FUNCTION_BLOCK FB_Tool EXTENDS FB_Base
VAR_INPUT
	sOpen: Skill_Greifer_open;
END_VAR
VAR_OUTPUT
	visStatus: stVisStatusTool;
END_VAR
VAR
END_VAR

ACTION CYCLIC_TOOL:
CYCLIC_BASE();


//VISSTATUS
//TODO

// GO INTO GREIFER.... INSTANCE OF THIS FB //todo
pA_Skills[1]:=ADR(sOpen);
sOpen(pTool:=THIS,pin:=9);
END_ACTION

METHOD PROTECTED onActivate : eResult
onActivate := eResult.SUCCESS;
      RETURN;
      // ---- Init ----
_transitionresult:=eResult.None;



// ---- Change ----

// _mode:= eMode.Automatic;




// ---- Check ----
_transitionresult := eResult.SUCCESS;


// ---- Change State ----
IF _transitionresult= eResult.SUCCESS THEN
	State:=eState.Active;
ELSIF _transitionresult= eResult.FAILURE THEN
	State:=eState.Inactive;
ELSIF _transitionresult= eResult.ERROR THEN
	State:=eState.ErrorProcessing;
ELSE
	ADSLOGSTR(ADSLOG_MSGTYPE_WARN,'Transitionresult from onActivate is None','');
END_IF
END_METHOD

METHOD PROTECTED onCleanup : eResult
onCleanup := eResult.SUCCESS;
      RETURN;
      // ---- Init ----
_transitionresult:=eResult.None;



// ---- Change ----

// _mode:= eMode.Manual;




// ---- Check ----
_transitionresult := eResult.SUCCESS;


// ---- Change State ----
IF _transitionresult= eResult.SUCCESS THEN
	State:=eState.Unconfigured;
ELSIF _transitionresult= eResult.FAILURE THEN
	ADSLOGSTR(ADSLOG_MSGTYPE_WARN,'Transitionresult from onCleanup is FAILURE ','');
ELSIF _transitionresult= eResult.ERROR THEN
	State:=eState.ErrorProcessing;
ELSE
	ADSLOGSTR(ADSLOG_MSGTYPE_WARN,'Transitionresult from onCleanup is NONE','');
END_IF
END_METHOD

METHOD PROTECTED onConfigure : eResult
onConfigure := eResult.SUCCESS;
      RETURN;
      // ---- Init ----
_transitionresult:=eResult.None;



// ---- Change ----

// _mode:= eMode.Manual;




// ---- Check ----
_transitionresult := eResult.SUCCESS;


// ---- Change State ----
IF _transitionresult= eResult.SUCCESS THEN
	State:=eState.Inactive;
ELSIF _transitionresult= eResult.FAILURE THEN
	State:=eState.Unconfigured;
ELSIF _transitionresult= eResult.ERROR THEN
	State:=eState.ErrorProcessing;
ELSE
	ADSLOGSTR(ADSLOG_MSGTYPE_WARN,'Transitionresult from onConfigure is None','');
END_IF
END_METHOD

METHOD PROTECTED onDeactivate : eResult
onDeactivate := eResult.SUCCESS;
      RETURN;
      // ---- Init ----
_transitionresult:=eResult.None;



// ---- Change ----

// _mode:= eMode.Manual;




// ---- Check ----
_transitionresult := eResult.SUCCESS;


// ---- Change State ----
IF _transitionresult= eResult.SUCCESS THEN
	State:=eState.Inactive;
ELSIF _transitionresult= eResult.FAILURE THEN
	ADSLOGSTR(ADSLOG_MSGTYPE_WARN,'Transitionresult from onDeactivate is FAILURE','');
ELSIF _transitionresult= eResult.ERROR THEN
	State:=eState.ErrorProcessing;
ELSE
	ADSLOGSTR(ADSLOG_MSGTYPE_WARN,'Transitionresult from onDeactivate is None','');
END_IF
END_METHOD

METHOD PROTECTED onError : eResult
onError := eResult.SUCCESS;
      RETURN;
      // ---- Init ----
_transitionresult:=eResult.None;



// ---- Change ----

// _mode:= eMode.Manual;




// ---- Check ----
_transitionresult := eResult.SUCCESS;


// ---- Change State ----
IF _transitionresult= eResult.SUCCESS THEN
	State:=eState.Unconfigured;
ELSIF _transitionresult= eResult.FAILURE THEN
	State:=eState.Finalized;
ELSIF _transitionresult= eResult.ERROR THEN
	ADSLOGSTR(ADSLOG_MSGTYPE_WARN,'Transitionresult from onError is Error','');
ELSE
	ADSLOGSTR(ADSLOG_MSGTYPE_WARN,'Transitionresult from onError is None','');
END_IF
END_METHOD

METHOD PROTECTED onShutdown : eResult
onShutdown := eResult.SUCCESS;
      RETURN;
      // ---- Init ----
_transitionresult:=eResult.None;



// ---- Change ----

// _mode:= eMode.Manual;




// ---- Check ----
_transitionresult := eResult.SUCCESS;


// ---- Change State ----
IF _transitionresult= eResult.SUCCESS THEN
	State:=eState.Finalized;
ELSIF _transitionresult= eResult.FAILURE THEN
	ADSLOGSTR(ADSLOG_MSGTYPE_WARN,'Transitionresult from onShutdown is FAILURE','');
ELSIF _transitionresult= eResult.ERROR THEN
	State:=eState.ErrorProcessing;
ELSE
	ADSLOGSTR(ADSLOG_MSGTYPE_WARN,'Transitionresult from onShutdown is None','');
END_IF
END_METHOD

END_FUNCTION_BLOCK

(* stored: Version 1.1.0.1, ProductVersion 3.1.4026.18
   POU FB_Tool: Id {b1d965f9-80c9-4ed1-8c86-7d42c5c70293}, SpecialFunc None
   Folder StateControl: Id {53ff33b6-3262-41f7-b537-f1feb7ee1671}
   Action CYCLIC_TOOL: Id {dff3f002-2f5f-470a-8757-89415d48f543}
   Method onActivate: Id {f08f7dc1-202a-4da9-a3e3-b4c98ccb8fdb}
   Method onCleanup: Id {5f653bd9-79a9-457e-9486-5b597592962d}
   Method onConfigure: Id {dbe1a2e7-a092-4589-85e0-cae2ad014539}
   Method onDeactivate: Id {7bafeac5-ea48-4fa6-837b-172e23cfe7dd}
   Method onError: Id {a42923bc-a704-4471-bfcc-ef605c0e08f9}
   Method onShutdown: Id {d564eedf-30cf-49ef-bdf9-182cbaf13e45} *)
